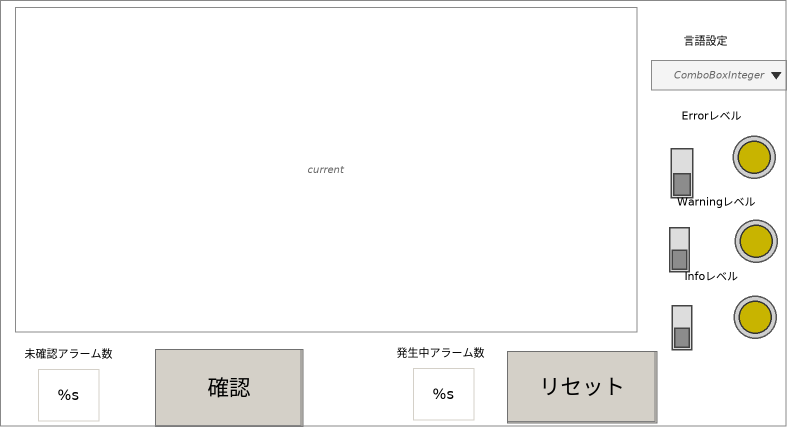
VISUALIZATION Visualization  // 787x427
    Button (155,349 148x78), "確認", colour toggle: MAIN.status_unconfirm
        tap MAIN.confirm_button_input
    DipSwitch (657,145 50x56), variable: MAIN.is_error, behaviour: TOGGLE, style: Switch-DipSwitch-Gray
    Button (507,351 150x72), "リセット", colour toggle: MAIN.status_resetable
        tap MAIN.reset_button_input
    DipSwitch (656,227 47x45), variable: MAIN.is_warning, behaviour: TOGGLE, style: Switch-DipSwitch-Gray
    DipSwitch (656,305 52x45), variable: MAIN.is_info, behaviour: TOGGLE, style: Switch-DipSwitch-Gray
    Lamp1 (729,131 50x52), variable: MAIN.is_error, style: Lamp-Lamp1-Yellow
    Lamp1 (731,215 50x52), variable: MAIN.is_warning, style: Lamp-Lamp1-Yellow
    Lamp1 (730,291 50x52), variable: MAIN.is_info, style: Lamp-Lamp1-Yellow
    Label (670,99 83x34), "Errorレベル"
    Label (675,185 83x34), "Warningレベル"
    Label (670,265 83x23), "Infoレベル"
    Textfield (38,369 61x52), "%s", text variable: MAIN.unconfirmed_count
    Textfield (413,368 61x52), "%s", text variable: MAIN.active_count
    Label (384,338 113x30), "発生中アラーム数"
    Label (12,339 113x30), "未確認アラーム数"
    TabControl (15,7 622x325)
        shows current()
        shows history()
        [0]: TabTitle=現在
        [1]: TabTitle=履歴
    Label (664,24 83x34), "言語設定"
    ComboBoxInteger (651,60 136x30), variable: MAIN.lang_select_options, text list: 'languages'
END_VISUALIZATION

(* stored: Version 1.1.0.1, ProductVersion 3.1.4024.15
   Visu Visualization: Id {230483c7-8b30-4964-94b1-66195911bb3b} *)
